{attribute 'qualified_only'}
{attribute 'strict'}
TYPE E_ComponentType :
(
	eComponentType_driver,
	eComponentType_axis,
	eComponentType_stateMachine,
	eComponentType_station,
	eComponentType_handler,
	eComponentType_Furnace
);
END_TYPE

(* stored: Version 1.1.0.1
   DUT E_ComponentType: Id {a6226614-f901-4bea-95f6-3439d5609300} *)
